FUNCTION F_FIFO_WRITE : BOOL
VAR_INPUT
	cbData : UDINT;
	pData : POINTER TO BYTE;
	
	cbBuffer : UDINT;
	pBuffer : POINTER TO BYTE;
END_VAR
VAR
END_VAR



FW_MemMove(pDest := pBuffer + cbData, pSrc := pBuffer, cbLen := cbBuffer - cbData);


FW_MemMove(pDest := pBuffer, pSrc := pData, cbLen := cbData);

END_FUNCTION

(* stored: Version 1.1.0.1, ProductVersion 3.1.4024.11
   POU F_FIFO_WRITE: Id {73b02f33-c1e4-40c7-9042-5e4e806ffcbe}, SpecialFunc None *)
